// TIA Portal V19 export
FUNCTION_BLOCK "Main_Safety_RTG1"   // FB123, F_FBD
{ S7_Optimized_Access := 'TRUE' }
// stored: AutoNumber false
BEGIN
END_FUNCTION_BLOCK
